(* CoDeSys 2.3 export: load_prm_test.exp *)

(* POU load_prmConfig_sp, ST *)
PROGRAM load_prmConfig_sp
""")
outfile.write("CASE prmID OF/n")

END_PROGRAM
